Staubli VAL3: clkValve10.pgx

program clkValve10()
begin
  call toggleValve(10)
end
